KUKA KRL program: ab_a_stb_st01_g08.src, ab_a_stb_st01_g08.dat

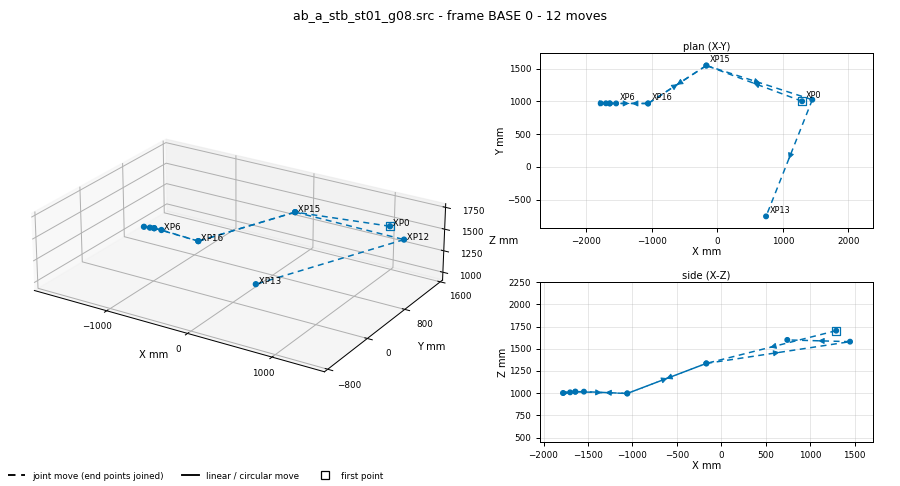
[picture p0: tool path of ab_a_stb_st01_g08.src in frame BASE 0, 12 of 12 moves have a stored position in this frame; points joined in program order, loops and branches not executed]
--- ab_a_stb_st01_g08.src ---
&ACCESS RV3
&REL 26
&PARAM DISKPATH = KRC:\R1\Program\MANIPULACAO NTC
DEF ab_a_stb_st01_g08( )
;FOLD INI;%{PE}
  ;FOLD BASISTECH INI
    GLOBAL INTERRUPT DECL 3 WHEN $STOPMESS==TRUE DO IR_STOPM ( )
    INTERRUPT ON 3
    BAS (#INITMOV,0 )
  ;ENDFOLD (BASISTECH INI)
;FOLD SPOTTECH INI
USERSPOT(#INIT)
;ENDFOLD (SPOTTECH INI)
;FOLD GRIPPERTECH INI
USER_GRP(0,DUMMY,DUMMY,GDEFAULT)
;ENDFOLD (GRIPPERTECH INI)
  ;FOLD USER INI
    ;Make your modifications here

  ;ENDFOLD (USER INI)
;ENDFOLD (INI)

; Caracterizacao dos meios de producao
; Changes: Deposita na Geo - Atego STB
; Versao Atual: 07/04/2016
; Ferramenta: GRIPPER ATEGO/AXOR
; Name: P13.090-R6

chk_w5_wechs_ok ( )  ; CHECK GRP ATEGO

chk_w5_grp1_opn ()
chk_w5_grp2_opn ()
chk_w5_grp3_opn ()
chk_w5_grp4_opn ()


;FOLD WAIT FOR ( NOT IN 497 'Presenca peca 1 Axor/Atego' );%{PE}%R 8.2.24,%MKUKATPBASIS,%CEXT_WAIT_FOR,%VEXT_WAIT_FOR,%P 2:, 4:NOT, 5:$IN, 6:497, 7:Presenca peca 1 Axor/Atego, 9:
WAIT FOR  (  NOT $IN[497] )
;ENDFOLD
;FOLD WAIT FOR ( NOT IN 498 'Presenca peca 2 Axor/Atego' );%{PE}%R 8.2.24,%MKUKATPBASIS,%CEXT_WAIT_FOR,%VEXT_WAIT_FOR,%P 2:, 4:NOT, 5:$IN, 6:498, 7:Presenca peca 2 Axor/Atego, 9:
WAIT FOR  (  NOT $IN[498] )
;ENDFOLD

;FOLD OUT 3347 'MAGAZINE 1 OCUPADO' State=TRUE ;%{PE}%R 8.2.24,%MKUKATPBASIS,%COUT,%VOUTX,%P 2:3347, 3:MAGAZINE 1 OCUPADO, 5:TRUE, 6:
$OUT[3347]=TRUE
;ENDFOLD
;FOLD OUT 3344 'APLICAÇÃO NÃO OK' State=TRUE ;%{PE}%R 8.2.24,%MKUKATPBASIS,%COUT,%VOUTX,%P 2:3344, 3:APLICAÇÃO NÃO OK, 5:TRUE, 6:
$OUT[3344]=TRUE
;ENDFOLD
;FOLD WAIT FOR ( IN 3347 'LIB. ANTECIPACAO (ATEGO/AXOR)' );%{PE}%R 8.2.24,%MKUKATPBASIS,%CEXT_WAIT_FOR,%VEXT_WAIT_FOR,%P 2:, 4:, 5:$IN, 6:3347, 7:LIB. ANTECIPACAO (ATEGO/AXOR), 9:
WAIT FOR  ( $IN[3347] )
;ENDFOLD
;FOLD OUT 3347 'MAGAZINE 1 OCUPADO' State=FALSE ;%{PE}%R 8.2.24,%MKUKATPBASIS,%COUT,%VOUTX,%P 2:3347, 3:MAGAZINE 1 OCUPADO, 5:FALSE, 6:
$OUT[3347]=FALSE
;ENDFOLD

;FOLD PTP P0 CONT Vel=100 % PDAT0 Tool[5]:Gripper Geo G01 00 Base[0];%{PE}%R 8.2.24,%MKUKATPBASIS,%CMOVE,%VPTP,%P 1:PTP, 2:P0, 3:C_PTP, 5:100, 7:PDAT0
$BWDSTART=FALSE
PDAT_ACT=PPDAT0
FDAT_ACT=FP0
BAS(#PTP_PARAMS,100)
PTP XP0 C_PTP
;ENDFOLD
;FOLD PTP P15 CONT Vel=100 % PDAT11 Tool[5]:Gripper Geo G01 00 Base[0];%{PE}%R 8.2.24,%MKUKATPBASIS,%CMOVE,%VPTP,%P 1:PTP, 2:P15, 3:C_PTP, 5:100, 7:PDAT11
$BWDSTART=FALSE
PDAT_ACT=PPDAT11
FDAT_ACT=FP15
BAS(#PTP_PARAMS,100)
PTP XP15 C_PTP
;ENDFOLD
;FOLD PTP P16 CONT Vel=100 % P_OLP7 Tool[5]:Gripper Geo G01 00 Base[0];%{PE}%R 8.2.24,%MKUKATPBASIS,%CMOVE,%VPTP,%P 1:PTP, 2:P16, 3:C_PTP, 5:100, 7:P_OLP7
$BWDSTART=FALSE
PDAT_ACT=PP_OLP7
FDAT_ACT=FP16
BAS(#PTP_PARAMS,100)
PTP XP16 C_PTP
;ENDFOLD

;FOLD WAIT FOR ( IN 3344 'LIB.P/APOIO DO TETO (ATEGO/AXOR)' );%{PE}%R 8.2.24,%MKUKATPBASIS,%CEXT_WAIT_FOR,%VEXT_WAIT_FOR,%P 2:, 4:, 5:$IN, 6:3344, 7:LIB.P/APOIO DO TETO (ATEGO/AXOR), 9:
WAIT FOR  ( $IN[3344] )
;ENDFOLD
;FOLD OUT 3344 'APLICAÇÃO NÃO OK' State=FALSE ;%{PE}%R 8.2.24,%MKUKATPBASIS,%COUT,%VOUTX,%P 2:3344, 3:APLICAÇÃO NÃO OK, 5:FALSE, 6:
$OUT[3344]=FALSE
;ENDFOLD

;FOLD PTP P6 CONT Vel=100 % PDAT6 Tool[5]:Gripper Geo G01 00 Base[0];%{PE}%R 8.2.24,%MKUKATPBASIS,%CMOVE,%VPTP,%P 1:PTP, 2:P6, 3:C_PTP, 5:100, 7:PDAT6
$BWDSTART=FALSE
PDAT_ACT=PPDAT6
FDAT_ACT=FP6
BAS(#PTP_PARAMS,100)
PTP XP6 C_PTP
;ENDFOLD
;FOLD LIN P7 CONT Vel=2 m/s CPDAT1 Tool[5]:Gripper Geo G01 00 Base[0];%{PE}%R 8.2.24,%MKUKATPBASIS,%CMOVE,%VLIN,%P 1:LIN, 2:P7, 3:C_DIS, 5:2, 7:CPDAT1
$BWDSTART=FALSE
LDAT_ACT=LCPDAT1
FDAT_ACT=FP7
BAS(#CP_PARAMS,2)
LIN XP7 C_DIS
;ENDFOLD
;FOLD LIN P17 CONT Vel=2 m/s CPDAT5 Tool[5]:Gripper Geo G01 00 Base[0];%{PE}%R 8.2.24,%MKUKATPBASIS,%CMOVE,%VLIN,%P 1:LIN, 2:P17, 3:C_DIS, 5:2, 7:CPDAT5
$BWDSTART=FALSE
LDAT_ACT=LCPDAT5
FDAT_ACT=FP17
BAS(#CP_PARAMS,2)
LIN XP17 C_DIS
;ENDFOLD

;FOLD ; Ponto de Geometria;%{PE}%R 8.2.24,%MKUKATPBASIS,%CCOMMENT,%VNORMAL,%P 2:Ponto  de  Geometria
;ENDFOLD
;FOLD LIN P8 Vel=0.25 m/s CPDAT2 Tool[5]:Gripper Geo G01 00 Base[0];%{PE}%R 8.2.24,%MKUKATPBASIS,%CMOVE,%VLIN,%P 1:LIN, 2:P8, 3:, 5:0.25, 7:CPDAT2
$BWDSTART=FALSE
LDAT_ACT=LCPDAT2
FDAT_ACT=FP8
BAS(#CP_PARAMS,0.25)
LIN XP8
;ENDFOLD

;FOLD ; ROBO EM POSICAO/GARRA DO FRONTAL;%{PE}%R 8.2.24,%MKUKATPBASIS,%CCOMMENT,%VNORMAL,%P 2:ROBO  EM  POSICAO/GARRA  DO  FRONTAL
;ENDFOLD
;FOLD OUT 3348 'STATUS DA SAIDA' State=TRUE ;%{PE}%R 8.2.24,%MKUKATPBASIS,%COUT,%VOUTX,%P 2:3348, 3:STATUS DA SAIDA, 5:TRUE, 6:
$OUT[3348]=TRUE
;ENDFOLD

;FOLD WAIT FOR ( IN 3348 'LIBERACAO FECHAR GRAMPOS/FRONTAL' );%{PE}%R 8.2.24,%MKUKATPBASIS,%CEXT_WAIT_FOR,%VEXT_WAIT_FOR,%P 2:, 4:, 5:$IN, 6:3348, 7:LIBERACAO FECHAR GRAMPOS/FRONTAL, 9:
WAIT FOR  ( $IN[3348] )
;ENDFOLD
;FOLD OUT 3348 'STATUS DA SAIDA' State=FALSE ;%{PE}%R 8.2.24,%MKUKATPBASIS,%COUT,%VOUTX,%P 2:3348, 3:STATUS DA SAIDA, 5:FALSE, 6:
$OUT[3348]=FALSE
;ENDFOLD

;FOLD ; Fechar grampos Z4;%{PE}%R 8.2.24,%MKUKATPBASIS,%CCOMMENT,%VNORMAL,%P 2:Fechar  grampos  Z4
;ENDFOLD
;FOLD SET GRP 4 State=CLO GDAT8;%{PE}%R 8.2.4,%MKUKATPGRP,%CGRP,%VGRP,%P 2:4, 4:1, 5:#NO, 6:GDAT8, 8:0, 10:0
H50(GRP,4,1,GGDAT8)
;ENDFOLD
;FOLD ; checar grampos Z4 fechados;%{PE}%R 8.2.24,%MKUKATPBASIS,%CCOMMENT,%VNORMAL,%P 2:checar  grampos  Z4  fechados
;ENDFOLD
chk_w5_grp4_clo ()

;FOLD ; Fechar grampos Z1 e Z2;%{PE}%R 8.2.24,%MKUKATPBASIS,%CCOMMENT,%VNORMAL,%P 2:Fechar  grampos  Z1  e  Z2
;ENDFOLD
;FOLD SET GRP 1 State=CLO GDAT6;%{PE}%R 8.2.4,%MKUKATPGRP,%CGRP,%VGRP,%P 2:1, 4:1, 5:#NO, 6:GDAT6, 8:0, 10:0
H50(GRP,1,1,GGDAT6)
;ENDFOLD
;FOLD SET GRP 2 State=CLO GDAT7;%{PE}%R 8.2.4,%MKUKATPGRP,%CGRP,%VGRP,%P 2:2, 4:1, 5:#NO, 6:GDAT7, 8:0, 10:0
H50(GRP,2,1,GGDAT7)
;ENDFOLD
;FOLD ; checar grampos Z1 e Z2 fechados;%{PE}%R 8.2.24,%MKUKATPBASIS,%CCOMMENT,%VNORMAL,%P 2:checar  grampos  Z1  e  Z2  fechados
;ENDFOLD
chk_w5_grp1_clo ()
chk_w5_grp2_clo ()

;FOLD ; Fechar grampos Z3;%{PE}%R 8.2.24,%MKUKATPBASIS,%CCOMMENT,%VNORMAL,%P 2:Fechar  grampos  Z3
;ENDFOLD
;FOLD SET GRP 3 State=CLO GDAT9;%{PE}%R 8.2.4,%MKUKATPGRP,%CGRP,%VGRP,%P 2:3, 4:1, 5:#NO, 6:GDAT9, 8:0, 10:0
H50(GRP,3,1,GGDAT9)
;ENDFOLD
;FOLD ; checar grampos Z3 fechados;%{PE}%R 8.2.24,%MKUKATPBASIS,%CCOMMENT,%VNORMAL,%P 2:checar  grampos  Z3  fechados
;ENDFOLD
chk_w5_grp3_clo ()

;FOLD ; Verifica garra com peca;%{PE}%R 8.2.24,%MKUKATPBASIS,%CCOMMENT,%VNORMAL,%P 2:Verifica  garra  com  peca
;ENDFOLD
IF (NOT(GHOST())) THEN
;FOLD WAIT FOR ( IN 497 'Presenca peca 1 Axor/Atego' );%{PE}%R 8.2.24,%MKUKATPBASIS,%CEXT_WAIT_FOR,%VEXT_WAIT_FOR,%P 2:, 4:, 5:$IN, 6:497, 7:Presenca peca 1 Axor/Atego, 9:
WAIT FOR  ( $IN[497] )
;ENDFOLD
;FOLD WAIT FOR ( IN 498 'Presenca peca 2 Axor/Atego' );%{PE}%R 8.2.24,%MKUKATPBASIS,%CEXT_WAIT_FOR,%VEXT_WAIT_FOR,%P 2:, 4:, 5:$IN, 6:498, 7:Presenca peca 2 Axor/Atego, 9:
WAIT FOR  ( $IN[498] )
;ENDFOLD
ENDIF

;FOLD ; Robo na posicao;%{PE}%R 8.2.24,%MKUKATPBASIS,%CCOMMENT,%VNORMAL,%P 2:Robo  na  posicao
;ENDFOLD
;FOLD OUT 3345 'ALERTA DE APLICAÇÃO' State=TRUE ;%{PE}%R 8.2.24,%MKUKATPBASIS,%COUT,%VOUTX,%P 2:3345, 3:ALERTA DE APLICAÇÃO, 5:TRUE, 6:
$OUT[3345]=TRUE
;ENDFOLD
;FOLD ; Aguarda liberacao para sair com a garra;%{PE}%R 8.2.24,%MKUKATPBASIS,%CCOMMENT,%VNORMAL,%P 2:Aguarda  liberacao  para  sair  com  a  garra
;ENDFOLD
;FOLD WAIT FOR ( IN 3345 'LIB.SAÍDA APOIO DO TETO (ATEGO/AXOR)' );%{PE}%R 8.2.24,%MKUKATPBASIS,%CEXT_WAIT_FOR,%VEXT_WAIT_FOR,%P 2:, 4:, 5:$IN, 6:3345, 7:LIB.SAÍDA APOIO DO TETO (ATEGO/AXOR), 9:
WAIT FOR  ( $IN[3345] )
;ENDFOLD
;FOLD OUT 3345 'ALERTA DE APLICAÇÃO' State=FALSE ;%{PE}%R 8.2.24,%MKUKATPBASIS,%COUT,%VOUTX,%P 2:3345, 3:ALERTA DE APLICAÇÃO, 5:FALSE, 6:
$OUT[3345]=FALSE
;ENDFOLD

;FOLD ; Abrir grampos Z1,Z2,Z4;%{PE}%R 8.2.24,%MKUKATPBASIS,%CCOMMENT,%VNORMAL,%P 2:Abrir  grampos  Z1,Z2,Z4
;ENDFOLD
;FOLD SET GRP 1 State=OPN GDAT2;%{PE}%R 8.2.4,%MKUKATPGRP,%CGRP,%VGRP,%P 2:1, 4:2, 5:#NO, 6:GDAT2, 8:0, 10:0
H50(GRP,1,2,GGDAT2)
;ENDFOLD
;FOLD SET GRP 2 State=OPN GDAT4;%{PE}%R 8.2.4,%MKUKATPGRP,%CGRP,%VGRP,%P 2:2, 4:2, 5:#NO, 6:GDAT4, 8:0, 10:0
H50(GRP,2,2,GGDAT4)
;ENDFOLD
;FOLD SET GRP 3 State=OPN GDAT5;%{PE}%R 8.2.4,%MKUKATPGRP,%CGRP,%VGRP,%P 2:3, 4:2, 5:#NO, 6:GDAT5, 8:0, 10:0
H50(GRP,3,2,GGDAT5)
;ENDFOLD
;FOLD SET GRP 4 State=OPN GDAT10;%{PE}%R 8.2.4,%MKUKATPGRP,%CGRP,%VGRP,%P 2:4, 4:2, 5:#NO, 6:GDAT10, 8:0, 10:0
H50(GRP,4,2,GGDAT10)
;ENDFOLD

chk_w5_grp1_opn ()
chk_w5_grp2_opn ()
chk_w5_grp3_opn ()
chk_w5_grp4_opn ()

;FOLD LIN P9 Vel=0.25 m/s CPDAT3 Tool[5]:Gripper Geo G01 00 Base[0];%{PE}%R 8.2.24,%MKUKATPBASIS,%CMOVE,%VLIN,%P 1:LIN, 2:P9, 3:, 5:0.25, 7:CPDAT3
$BWDSTART=FALSE
LDAT_ACT=LCPDAT3
FDAT_ACT=FP9
BAS(#CP_PARAMS,0.25)
LIN XP9
;ENDFOLD

;FOLD ; Verifica garra sem peca;%{PE}%R 8.2.24,%MKUKATPBASIS,%CCOMMENT,%VNORMAL,%P 2:Verifica  garra  sem  peca
;ENDFOLD
;FOLD WAIT FOR ( NOT IN 497 'Presenca peca 1 Axor/Atego' );%{PE}%R 8.2.24,%MKUKATPBASIS,%CEXT_WAIT_FOR,%VEXT_WAIT_FOR,%P 2:, 4:NOT, 5:$IN, 6:497, 7:Presenca peca 1 Axor/Atego, 9:
WAIT FOR  (  NOT $IN[497] )
;ENDFOLD
;FOLD WAIT FOR ( NOT IN 498 'Presenca peca 2 Axor/Atego' );%{PE}%R 8.2.24,%MKUKATPBASIS,%CEXT_WAIT_FOR,%VEXT_WAIT_FOR,%P 2:, 4:NOT, 5:$IN, 6:498, 7:Presenca peca 2 Axor/Atego, 9:
WAIT FOR  (  NOT $IN[498] )
;ENDFOLD

;FOLD PTP P10 CONT Vel=100 % PDAT7 Tool[5]:Gripper Geo G01 00 Base[0];%{PE}%R 8.2.24,%MKUKATPBASIS,%CMOVE,%VPTP,%P 1:PTP, 2:P10, 3:C_PTP, 5:100, 7:PDAT7
$BWDSTART=FALSE
PDAT_ACT=PPDAT7
FDAT_ACT=FP10
BAS(#PTP_PARAMS,100)
PTP XP10 C_PTP
;ENDFOLD
;FOLD PTP P11 Vel=100 % PDAT8 Tool[5]:Gripper Geo G01 00 Base[0];%{PE}%R 8.2.24,%MKUKATPBASIS,%CMOVE,%VPTP,%P 1:PTP, 2:P11, 3:, 5:100, 7:PDAT8
$BWDSTART=FALSE
PDAT_ACT=PPDAT8
FDAT_ACT=FP11
BAS(#PTP_PARAMS,100)
PTP XP11
;ENDFOLD

;FOLD ; Libera dispositivo para soldar Respot;%{PE}%R 8.2.24,%MKUKATPBASIS,%CCOMMENT,%VNORMAL,%P 2:Libera  dispositivo  para  soldar  Respot
;ENDFOLD
;FOLD OUT 3347 'MAGAZINE 1 OCUPADO' State=TRUE ;%{PE}%R 8.2.24,%MKUKATPBASIS,%COUT,%VOUTX,%P 2:3347, 3:MAGAZINE 1 OCUPADO, 5:TRUE, 6:
$OUT[3347]=TRUE
;ENDFOLD
;FOLD OUT 3344 'APLICAÇÃO NÃO OK' State=TRUE ;%{PE}%R 8.2.24,%MKUKATPBASIS,%COUT,%VOUTX,%P 2:3344, 3:APLICAÇÃO NÃO OK, 5:TRUE, 6:
$OUT[3344]=TRUE
;ENDFOLD

;FOLD PULSE 3340 'R6 GEOMETRIA OK' State=TRUE Time=1 sec;%{PE}%R 8.2.24,%MKUKATPBASIS,%COUT,%VPULSE,%P 2:3340, 3:R6 GEOMETRIA OK, 5:TRUE, 6:, 8:1
PULSE($OUT[3340], TRUE,1)
;ENDFOLD

;FOLD PTP P12 CONT Vel=100 % PDAT9 Tool[5]:Gripper Geo G01 00 Base[0];%{PE}%R 8.2.24,%MKUKATPBASIS,%CMOVE,%VPTP,%P 1:PTP, 2:P12, 3:C_PTP, 5:100, 7:PDAT9
$BWDSTART=FALSE
PDAT_ACT=PPDAT9
FDAT_ACT=FP12
BAS(#PTP_PARAMS,100)
PTP XP12 C_PTP
;ENDFOLD

;FOLD PTP P13 Vel=100 % PDAT10 Tool[5]:Gripper Geo G01 00 Base[0];%{PE}%R 8.2.24,%MKUKATPBASIS,%CMOVE,%VPTP,%P 1:PTP, 2:P13, 3:, 5:100, 7:PDAT10
$BWDSTART=FALSE
PDAT_ACT=PPDAT10
FDAT_ACT=FP13
BAS(#PTP_PARAMS,100)
PTP XP13
;ENDFOLD

END

--- ab_a_stb_st01_g08.dat ---
&ACCESS RV3
&REL 26
&PARAM DISKPATH = KRC:\R1\Program\MANIPULACAO NTC
DEFDAT  ab_a_stb_st01_g08
;FOLD EXTERNAL DECLARATIONS;%{PE}%MKUKATPBASIS,%CEXT,%VCOMMON,%P
;FOLD BASISTECH EXT;%{PE}%MKUKATPBASIS,%CEXT,%VEXT,%P
EXT  BAS (BAS_COMMAND  :IN,REAL  :IN )
DECL INT SUCCESS
;ENDFOLD (BASISTECH EXT)
;FOLD USER EXT;%{E}%MKUKATPUSER,%CEXT,%VEXT,%P
;Make your modifications here
;ENDFOLD (USER EXT)
;ENDFOLD (EXTERNAL DECLARATIONS)

;# ============ START PATH : ab_a_stb_st01_g08 =============
DECL FDAT Fp111={TOOL_NO 5,BASE_NO 0,IPO_FRAME #BASE,POINT2[] " "}
DECL PDAT PP_OLP1={VEL 100.0,ACC 100.0,APO_DIST 0.0}
DECL E6POS Xp111={X 1293.05298,Y 1000.52002,Z 1703.34204,A 36.1688995,B -6.95510006,C 153.792694,S 6,T 19}
DECL FDAT Fp110={TOOL_NO 5,BASE_NO 0,IPO_FRAME #BASE,POINT2[] " "}
DECL PDAT PP_OLP2={VEL 100.0,ACC 100.0,APO_DIST 0.0}
DECL E6POS Xp110={X -168.237,Y 1546.06995,Z 1335.04004,A 110.0187,B -0.406599998,C 159.128998,S 6,T 19}
DECL FDAT Fp104={TOOL_NO 5,BASE_NO 0,IPO_FRAME #BASE,POINT2[] " "}
DECL PDAT PP_OLP3={VEL 100.0,ACC 100.0,APO_DIST 0.0}
DECL E6POS Xp104={X -1057.83704,Y 966.953003,Z 997.169983,A -179.672195,B -1.48539996,C 179.896301,S 6,T 19}
DECL FDAT Fp2={TOOL_NO 5,BASE_NO 0,IPO_FRAME #BASE,POINT2[] " ",TQ_STATE FALSE}
DECL E6POS Xp102={X -1642.28699,Y 967.63501,Z 1017.06799,A 179.793503,B -1.63569999,C 179.849304,S 6,T 19}
DECL LDAT LL_OLP1={VEL 2.0,ACC 100.0,APO_DIST 0.0,APO_FAC 0.0,ORI_TYP #VAR,CIRC_TYP #BASE,JERK_FAC 50.0}
DECL FDAT Fl005={TOOL_NO 5,BASE_NO 0,IPO_FRAME #BASE,POINT2[] " "}
DECL E6POS Xl005={X -1792.44604,Y 967.633972,Z 1017.06897,A 179.793503,B -1.63569999,C 179.849304,S 6,T 19}
DECL LDAT LL_OLP2={VEL 1.0,ACC 100.0,APO_DIST 0.0,APO_FAC 0.0,ORI_TYP #VAR,CIRC_TYP #BASE,JERK_FAC 50.0}
DECL FDAT Fp107={TOOL_NO 5,BASE_NO 0,IPO_FRAME #BASE,POINT2[] " "}
DECL E6POS Xp107={X -1642.28699,Y 967.63501,Z 1017.06799,A 179.793503,B -1.63569999,C 179.849304,S 6,T 19}
DECL LDAT LL_OLP3={VEL 0.25,ACC 100.0,APO_DIST 0.0,APO_FAC 0.0,ORI_TYP #VAR,CIRC_TYP #BASE,JERK_FAC 50.0}
DECL FDAT Fp108={TOOL_NO 5,BASE_NO 0,IPO_FRAME #BASE,POINT2[] " "}
DECL PDAT PP_OLP4={VEL 100.0,ACC 100.0,APO_DIST 0.0}
DECL E6POS Xp108={X -1057.83704,Y 966.952026,Z 997.169983,A -179.672195,B -1.48529994,C 179.896393,S 6,T 19}
DECL FDAT Fp109={TOOL_NO 5,BASE_NO 0,IPO_FRAME #BASE,POINT2[] " "}
DECL PDAT PP_OLP5={VEL 100.0,ACC 100.0,APO_DIST 0.0}
DECL E6POS Xp109={X -168.235992,Y 1546.07104,Z 1335.03699,A 110.0187,B -0.406500012,C 159.128998,S 6,T 19}
DECL FDAT Fp112={TOOL_NO 5,BASE_NO 0,IPO_FRAME #BASE,POINT2[] " "}
DECL PDAT PP_OLP6={VEL 100.0,ACC 100.0,APO_DIST 0.0}
DECL E6POS Xp112={X 1293.052,Y 1000.521,Z 1703.34302,A 36.1689987,B -6.95510006,C 153.792801,S 6,T 19}
DECL BASIS_SUGG_T LAST_BASIS={POINT1[] "P0                      ",POINT2[] "P0                      ",CP_PARAMS[] "CPDAT0                  ",PTP_PARAMS[] "PDAT0                   ",CONT[] "                        ",CP_VEL[] "2.0                     ",PTP_VEL[] " 100                    ",SYNC_PARAMS[] "SYNCDAT                 ",SPL_NAME[] "S0                      "}
DECL FDAT Fp102={TOOL_NO 5,BASE_NO 0,IPO_FRAME #BASE,POINT2[] " ",TQ_STATE FALSE}
DECL E6POS XP1={X 932.898682,Y -1400.41504,Z 2058.77808,A -72.0052567,B -60.9366112,C 178.901398,S 18,T 2,E1 0.0,E2 0.0,E3 0.0,E4 0.0,E5 0.0,E6 0.0}
DECL FDAT FP1={TOOL_NO 5,BASE_NO 0,IPO_FRAME #BASE,POINT2[] " ",TQ_STATE FALSE}
DECL PDAT PPDAT1={VEL 100.0,ACC 100.0,APO_DIST 100.0,GEAR_JERK 50.0}
DECL PDAT PPDAT2={VEL 100.0,ACC 20.0,APO_DIST 100.0,GEAR_JERK 50.0}
DECL E6POS XP2={X 742.641113,Y -756.368286,Z 1599.64197,A -36.0531006,B 42.8925095,C 82.0326691,S 18,T 2,E1 0.0,E2 0.0,E3 0.0,E4 0.0,E5 0.0,E6 0.0}
DECL E6POS XP3={X 1357.67297,Y -467.458099,Z 2426.61206,A 68.9576263,B 36.5581284,C 80.2279587,S 22,T 18,E1 0.0,E2 0.0,E3 0.0,E4 0.0,E5 0.0,E6 0.0}
DECL FDAT FP3={TOOL_NO 5,BASE_NO 0,IPO_FRAME #BASE,POINT2[] " ",TQ_STATE FALSE}
DECL PDAT PPDAT3={VEL 100.0,ACC 100.0,APO_DIST 100.0,APO_MODE #CPTP,GEAR_JERK 50.0}
DECL E6POS XP4={X 1293.13599,Y 1000.34998,Z 1703.13794,A 36.1652107,B -6.94713116,C 153.780899,S 22,T 19,E1 0.0,E2 0.0,E3 0.0,E4 0.0,E5 0.0,E6 0.0}
DECL FDAT FP4={TOOL_NO 5,BASE_NO 0,IPO_FRAME #BASE,POINT2[] " ",TQ_STATE FALSE}
DECL PDAT PPDAT4={VEL 100.0,ACC 20.0,APO_DIST 100.0,APO_MODE #CPTP,GEAR_JERK 50.0}
DECL E6POS XP5={X -168.100403,Y 1546.15405,Z 1334.922,A 110.012604,B -0.403610796,C 159.120895,S 22,T 19,E1 0.0,E2 0.0,E3 0.0,E4 0.0,E5 0.0,E6 0.0}
DECL FDAT FP5={TOOL_NO 5,BASE_NO 0,IPO_FRAME #BASE,POINT2[] " ",TQ_STATE FALSE}
DECL PDAT PPDAT5={VEL 100.0,ACC 20.0,APO_DIST 20.0,APO_MODE #CPTP,GEAR_JERK 50.0}
DECL E6POS XP6={X -1545.40405,Y 967.62738,Z 1017.44897,A 179.793198,B -1.63709199,C 179.851593,S 22,T 19,E1 0.0,E2 0.0,E3 0.0,E4 0.0,E5 0.0,E6 0.0}
DECL FDAT FP6={TOOL_NO 5,BASE_NO 0,IPO_FRAME #BASE,POINT2[] " ",TQ_STATE FALSE}
DECL PDAT PPDAT6={VEL 100.0,ACC 20.0,APO_DIST 100.0,APO_MODE #CPTP,GEAR_JERK 50.0}
DECL E6POS XP7={X -1642.27905,Y 967.633606,Z 1017.07202,A 179.793793,B -1.63576603,C 179.849701,S 22,T 19,E1 0.0,E2 0.0,E3 0.0,E4 0.0,E5 0.0,E6 0.0}
DECL FDAT FP7={TOOL_NO 5,BASE_NO 0,IPO_FRAME #BASE,POINT2[] " ",TQ_STATE FALSE}
DECL LDAT LCPDAT1={VEL 2.0,ACC 100.0,APO_DIST 100.0,APO_FAC 50.0,AXIS_VEL 100.0,AXIS_ACC 100.0,ORI_TYP #VAR,CIRC_TYP #BASE,JERK_FAC 50.0,GEAR_JERK 50.0,EXAX_IGN 0}
DECL E6POS XP8={X -1781.22998,Y 969.123901,Z 1001.77002,A 179.957703,B -0.387168914,C 179.691299,S 22,T 19,E1 0.0,E2 0.0,E3 0.0,E4 0.0,E5 0.0,E6 0.0}
DECL FDAT FP8={TOOL_NO 5,BASE_NO 0,IPO_FRAME #BASE,POINT2[] " ",TQ_STATE FALSE}
DECL LDAT LCPDAT2={VEL 2.0,ACC 100.0,APO_DIST 100.0,APO_FAC 50.0,AXIS_VEL 100.0,AXIS_ACC 100.0,ORI_TYP #VAR,CIRC_TYP #BASE,JERK_FAC 50.0,GEAR_JERK 50.0,EXAX_IGN 0}
DECL E6POS XP9={X -1642.26697,Y 967.633911,Z 1017.05701,A 179.794006,B -1.63522899,C 179.849197,S 22,T 19,E1 0.0,E2 0.0,E3 0.0,E4 0.0,E5 0.0,E6 0.0}
DECL FDAT FP9={TOOL_NO 5,BASE_NO 0,IPO_FRAME #BASE,POINT2[] " ",TQ_STATE FALSE}
DECL LDAT LCPDAT3={VEL 2.0,ACC 100.0,APO_DIST 100.0,APO_FAC 50.0,AXIS_VEL 100.0,AXIS_ACC 100.0,ORI_TYP #VAR,CIRC_TYP #BASE,JERK_FAC 50.0,GEAR_JERK 50.0,EXAX_IGN 0}
DECL E6POS XP10={X -1057.84595,Y 966.967773,Z 997.154419,A -179.673004,B -1.48506796,C 179.895401,S 22,T 19,E1 0.0,E2 0.0,E3 0.0,E4 0.0,E5 0.0,E6 0.0}
DECL FDAT FP10={TOOL_NO 5,BASE_NO 0,IPO_FRAME #BASE,POINT2[] " ",TQ_STATE FALSE}
DECL PDAT PPDAT7={VEL 100.0,ACC 20.0,APO_DIST 20.0,APO_MODE #CPTP,GEAR_JERK 50.0}
DECL E6POS XP11={X -168.311401,Y 1546.02295,Z 1335.104,A 110.022797,B -0.408378392,C 159.132599,S 22,T 19,E1 0.0,E2 0.0,E3 0.0,E4 0.0,E5 0.0,E6 0.0}
DECL FDAT FP11={TOOL_NO 5,BASE_NO 0,IPO_FRAME #BASE,POINT2[] " ",TQ_STATE FALSE}
DECL PDAT PPDAT8={VEL 100.0,ACC 20.0,APO_DIST 20.0,APO_MODE #CPTP,GEAR_JERK 50.0}
DECL E6POS XP12={X 1448.77295,Y 1024.36804,Z 1579.73096,A 38.2694511,B -5.98833799,C 154.415405,S 22,T 19,E1 0.0,E2 0.0,E3 0.0,E4 0.0,E5 0.0,E6 0.0}
DECL FDAT FP12={TOOL_NO 5,BASE_NO 0,IPO_FRAME #BASE,POINT2[] " ",TQ_STATE FALSE}
DECL PDAT PPDAT9={VEL 100.0,ACC 20.0,APO_DIST 20.0,APO_MODE #CPTP,GEAR_JERK 50.0}
DECL E6POS XP13={X 742.836609,Y -756.080078,Z 1599.49402,A -36.0376701,B 42.89188,C 82.0582962,S 18,T 2,E1 0.0,E2 0.0,E3 0.0,E4 0.0,E5 0.0,E6 0.0}
DECL FDAT FP13={TOOL_NO 5,BASE_NO 0,IPO_FRAME #BASE,POINT2[] " ",TQ_STATE FALSE}
DECL PDAT PPDAT10={VEL 100.0,ACC 20.0,APO_DIST 100.0,GEAR_JERK 50.0}
DECL GRP_SUGG_T LAST_GRP={NUMBER[] "4                       ",STATE[] "1                       ",PARAMS[] "GDAT1                   "}
DECL GRP_TYP GGDAT1={G_APO #NO,GRP_TIME 0.200000003,CTRL #OFF,DLY 0,DST 1}
DECL GRP_TYP GGDAT8={G_APO #NO,GRP_TIME 0.200000003,CTRL #OFF,DLY 0,DST 1}
DECL GRP_TYP GGDAT6={G_APO #NO,GRP_TIME 0.200000003,CTRL #OFF,DLY 0,DST 1}
DECL GRP_TYP GGDAT7={G_APO #NO,GRP_TIME 0.200000003,CTRL #OFF,DLY 0,DST 1}
DECL GRP_TYP GGDAT9={G_APO #NO,GRP_TIME 0.200000003,CTRL #OFF,DLY 0,DST 1}
DECL GRP_TYP GGDAT2={G_APO #NO,GRP_TIME 0.200000003,CTRL #OFF,DLY 0,DST 1}
DECL GRP_TYP GGDAT4={G_APO #NO,GRP_TIME 0.200000003,CTRL #OFF,DLY 0,DST 1}
DECL GRP_TYP GGDAT5={G_APO #NO,GRP_TIME 0.200000003,CTRL #OFF,DLY 0,DST 1}
DECL GRP_TYP GGDAT10={G_APO #NO,GRP_TIME 0.200000003,CTRL #OFF,DLY 0,DST 1}
DECL E6POS XP14={X -1783.76294,Y 971.845581,Z 1012.17499,A -179.926193,B -0.738284171,C 179.847198,S 22,T 19,E1 0.0,E2 0.0,E3 0.0,E4 0.0,E5 0.0,E6 0.0}
DECL FDAT FP14={TOOL_NO 5,BASE_NO 0,IPO_FRAME #BASE,POINT2[] " ",TQ_STATE FALSE}
DECL LDAT LCPDAT4={VEL 2.0,ACC 100.0,APO_DIST 100.0,APO_FAC 50.0,AXIS_VEL 100.0,AXIS_ACC 100.0,ORI_TYP #VAR,CIRC_TYP #BASE,JERK_FAC 50.0,GEAR_JERK 50.0,EXAX_IGN 0}
DECL PDAT PPDAT0={VEL 100.0,ACC 20.0,APO_DIST 20.0,APO_MODE #CPTP,GEAR_JERK 50.0}
DECL E6POS XP0={X 1293.05103,Y 1000.526,Z 1703.34595,A 36.1689301,B -6.95535898,C 153.792694,S 22,T 19,E1 0.0,E2 0.0,E3 0.0,E4 0.0,E5 0.0,E6 0.0}
DECL FDAT FP0={TOOL_NO 5,BASE_NO 0,IPO_FRAME #BASE,POINT2[] " ",TQ_STATE FALSE}
DECL PDAT PPDAT11={VEL 100.0,ACC 20.0,APO_DIST 20.0,APO_MODE #CPTP,GEAR_JERK 50.0}
DECL E6POS XP15={X -168.237503,Y 1546.06799,Z 1335.04297,A 110.018799,B -0.406741798,C 159.129105,S 22,T 19,E1 0.0,E2 0.0,E3 0.0,E4 0.0,E5 0.0,E6 0.0}
DECL FDAT FP15={TOOL_NO 5,BASE_NO 0,IPO_FRAME #BASE,POINT2[] " ",TQ_STATE FALSE}
DECL PDAT PP_OLP7={VEL 100.0,ACC 20.0,APO_DIST 0.0,APO_MODE #CPTP}
DECL E6POS XP16={X -1057.83704,Y 966.953003,Z 997.169983,A -179.672195,B -1.48539996,C 179.896301,S 6,T 19}
DECL FDAT FP16={TOOL_NO 5,BASE_NO 0,IPO_FRAME #BASE,POINT2[] " "}
DECL E6POS XP17={X -1700.90698,Y 969.437683,Z 1009.552,A 179.905701,B -1.26266694,C 179.786194,S 22,T 19,E1 0.0,E2 0.0,E3 0.0,E4 0.0,E5 0.0,E6 0.0}
DECL FDAT FP17={TOOL_NO 5,BASE_NO 0,IPO_FRAME #BASE,POINT2[] " ",TQ_STATE FALSE}
DECL LDAT LCPDAT5={VEL 2.0,ACC 100.0,APO_DIST 100.0,APO_FAC 50.0,AXIS_VEL 100.0,AXIS_ACC 100.0,ORI_TYP #VAR,CIRC_TYP #BASE,JERK_FAC 50.0,GEAR_JERK 50.0,EXAX_IGN 0}
ENDDAT
